Fanuc TP program (LS listing): Prog1.ls

/PROG  Prog1
/ATTR
OWNER       = MNEDITOR;
COMMENT     = "FermePince"
PROG_SIZE   = 913;
CREATE      = DATE 22-03-16  TIME 16:56:07;
MODIFIED      = DATE 22-03-16  TIME 16:56:07;
FILE_NAME   = ;
VERSION    = 0;
LINE_COUNT  = 13;
MEMORY_SIZE = 1197;
PROTECT     = READ_WRITE;
TCD:  STACK_SIZE    = 0,
      TASK_PRIORITY = 50,
      TIME_SLICE    = 0,
      BUSY_LAMP_OFF = 0,
      ABORT_REQUEST = 0,
      PAUSE_REQUEST = 0;
DEFAULT_GROUP   = 1,*,*,*,*,*,*,* ;
CONTROL_CODE    = 00000000 00000000;
/APPL
/MN
1:!FANUC Robotics America ;
2:!ROBOGUIDE Generated This TPP ;
3:!Run SimPRO.cf to setup frame and tool data ;
4:!This program will be overwritten on the next save or run. ;
/POS
/END
